// Mitsubishi GX Works2 project: FX1s-14MR-led   PLC: FX1S

PROGRAM MAIN
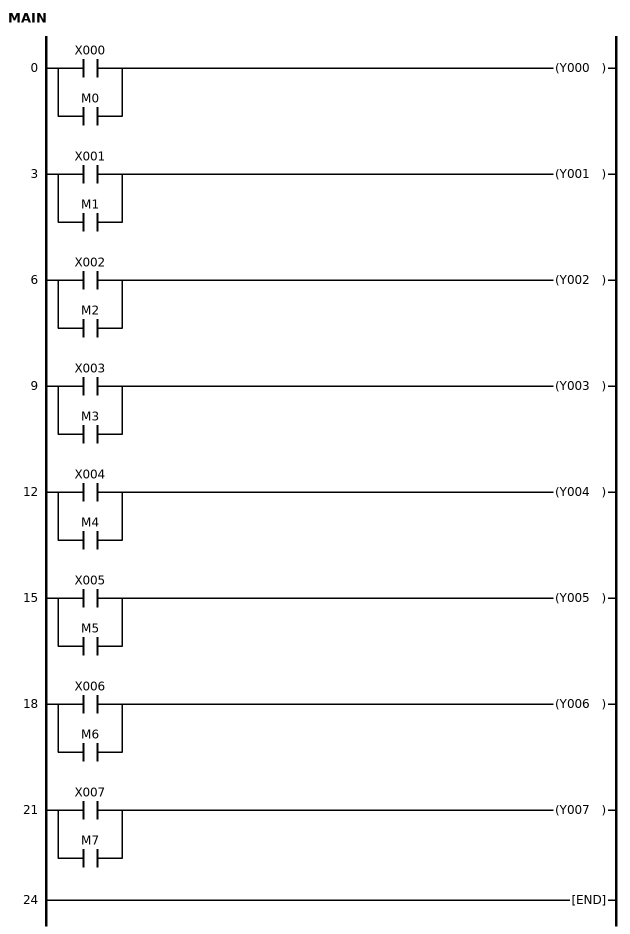
0     LD      X000
      OR      M0
      OUT     Y000
3     LD      X001
      OR      M1
      OUT     Y001
6     LD      X002
      OR      M2
      OUT     Y002
9     LD      X003
      OR      M3
      OUT     Y003
12    LD      X004
      OR      M4
      OUT     Y004
15    LD      X005
      OR      M5
      OUT     Y005
18    LD      X006
      OR      M6
      OUT     Y006
21    LD      X007
      OR      M7
      OUT     Y007
24    END
END_PROGRAM
